PROGRAM Q8
VAR
	input : BOOL;
	output: BOOL;
END_VAR

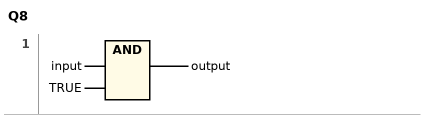
// NETWORK 1
output := input AND TRUE;

END_PROGRAM

(* stored: Version 1.1.0.1, ProductVersion 3.1.4024.12
   POU Q8: Id {107690a3-21af-4931-a969-a3e94b5a0643}, SpecialFunc None *)
